// TIA Portal project "ModbusTCP" (V19)

(* hardware
DEVICE "S7-1200 station_1"  S7-1200 Station
   slot 0: "Rack_0"  S7-1200 Rack  Rack  V1.0
   slot 1: "PLC_1"  CPU 1215C DC/DC/DC  6ES7 215-1AG40-0XB0  V4.6
*)

// ===== PLC "PLC_1"  CPU 1215C DC/DC/DC =====

VAR_GLOBAL   // PLC tag table "Default tag table"
   "Clock_Byte" AT %MB0 : Byte;
   "Clock_10Hz" AT %M0.0 : Bool;
   "Clock_5Hz" AT %M0.1 : Bool;
   "Clock_2.5Hz" AT %M0.2 : Bool;
   "Clock_2Hz" AT %M0.3 : Bool;
   "Clock_1.25Hz" AT %M0.4 : Bool;
   "Clock_1Hz" AT %M0.5 : Bool;
   "Clock_0.625Hz" AT %M0.6 : Bool;
   "Clock_0.5Hz" AT %M0.7 : Bool;
   "System_Byte" AT %MB1 : Byte;
   "FirstScan" AT %M1.0 : Bool;
   "DiagStatusUpdate" AT %M1.1 : Bool;
   "AlwaysTRUE" AT %M1.2 : Bool;
   "AlwaysFALSE" AT %M1.3 : Bool;
END_VAR

DATA_BLOCK "datosMB"   // DB1
{ S7_Optimized_Access := 'FALSE' }
VERSION : 0.1
   VAR
      Dato : Array[0..2] of Bool;
   END_VAR
BEGIN
END_DATA_BLOCK

DATA_BLOCK "connection"   // DB3
{ S7_Optimized_Access := 'TRUE' }
VERSION : 0.1
   VAR
      "Conexion 1" : TCON_IP_v4;
   END_VAR
BEGIN
   "Conexion 1".InterfaceId := 64;
   "Conexion 1".ID := 1;
   "Conexion 1".ConnectionType := 11;
   "Conexion 1".ActiveEstablished := true;
   "Conexion 1".RemoteAddress.ADDR[1] := 192;
   "Conexion 1".RemoteAddress.ADDR[2] := 168;
   "Conexion 1".RemoteAddress.ADDR[3] := 13;
   "Conexion 1".RemoteAddress.ADDR[4] := 63;
   "Conexion 1".RemotePort := 502;
END_DATA_BLOCK

ORGANIZATION_BLOCK "Main"   // OB1, LAD, ProgramCycle
TITLE = "Main Program Sweep (Cycle)"
{ S7_Optimized_Access := 'TRUE' }
VERSION : 0.1
   VAR_INPUT
      Initial_Call : Bool;   // Initial call of this OB
      Remanence : Bool;   // =True, if remanent data are available
   END_VAR
BEGIN

REGION Network 1
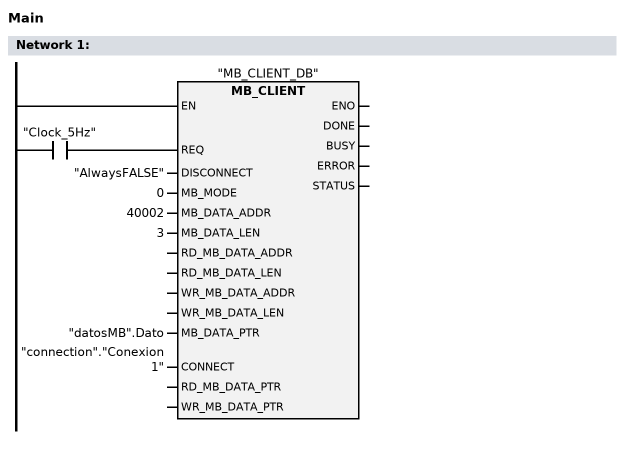
   "MB_CLIENT_DB"(REQ := "Clock_5Hz",   // MB_CLIENT
                  DISCONNECT := "AlwaysFALSE",
                  MB_MODE := 0,
                  MB_DATA_ADDR := 40002,
                  MB_DATA_LEN := 3,
                  MB_DATA_PTR := "datosMB".Dato,
                  CONNECT := "connection"."Conexion 1");
END_REGION
END_ORGANIZATION_BLOCK